// Mitsubishi GX Works2 project: 실습2인터록   PLC: Q02/Q02H

PROGRAM MAIN
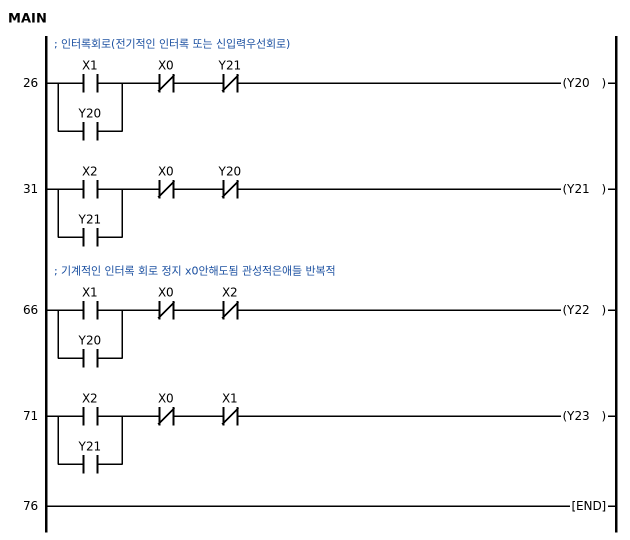
; 인터록회로(전기적인 인터록 또는 신입력우선회로)
26    LD      X1
      OR      Y20
      ANI     X0
      ANI     Y21
      OUT     Y20
31    LD      X2
      OR      Y21
      ANI     X0
      ANI     Y20
      OUT     Y21
; 기계적인 인터록 회로 정지 x0안해도됨 관성적은애들 반복적
66    LD      X1
      OR      Y20
      ANI     X0
      ANI     X2
      OUT     Y22
71    LD      X2
      OR      Y21
      ANI     X0
      ANI     X1
      OUT     Y23
76    END
END_PROGRAM
